FUNCTION F_PlatformAnglePos2CylPos : LREAL
VAR_INPUT
	fPlatformAngleTheta1Ref : LREAL;
END_VAR
VAR
	pi : LREAL := 3.14159265;
	fMinLengthPlatformCylinder : LREAL := 0.878;
	fOffsetAngleDeg : LREAL := 55.4;
	fOffsetAngleRad : LREAL	:= fOffsetAngleDeg*pi/180;
	fLengthA : LREAL	:= 0.513; 
	fLengthC : LREAL	:= 1.353; 
	fAngleBeta : LREAL;
	fCylinderLength : LREAL; 
END_VAR

fAngleBeta := fPlatformAngleTheta1Ref - fOffsetAngleRad;

fCylinderLength := SQRT(fLengthA*fLengthA + fLengthC*fLengthC - 2*fLengthA*fLengthC*COS(fAngleBeta));

F_PlatformAnglePos2CylPos := fCylinderLength - fMinLengthPlatformCylinder;

END_FUNCTION

(* stored: Version 1.1.0.1, ProductVersion 3.1.4024.12
   POU F_PlatformAnglePos2CylPos: Id {18b4b6cf-8455-42de-a342-c879dadc6a8a}, SpecialFunc None *)
